(* IEC 61131-3 sources: AXOpen/src/integrations/app/src/Examples/AXOpen.AxoTask, 2 files *)

(* ---- AxoTaskDocuExample.st ---- *)
USING AXOpen.Core;

NAMESPACE AxoTaskExamples
    {S7.extern=ReadWrite}
    CLASS AxoTaskDocuExample EXTENDS  AXOpen.Core.AxoContext
        VAR PUBLIC
            {#ix-set:AttributeName = "<#Task name#>"}
            _myTask : AxoTask;
            _myCounter : ULINT;
        END_VAR

        METHOD PUBLIC Initialize
            // Initialization of the context needs to be called first
            // It does not need to be called cyclically, just once
            THIS.InitializeRootObject(_myTask);
        END_METHOD

        METHOD PROTECTED OVERRIDE Main
            THIS.InitializeRootObject(_myTask);
            // Cyclicall call of the Execute
            IF _myTask.Execute() THEN
                _myCounter := _myCounter + ULINT#1;
                _myTask.DoneWhen(_myCounter = ULINT#100);
            END_IF;
            IF _myTask.IsDone() THEN
                _myCounter := ULINT#0;
            END_IF;
        END_METHOD

        METHOD Examples
        //<AxoTaskInvokeDone>
            IF _myTask.Invoke().IsDone() THEN
                ; //Do something
            END_IF;
        //</AxoTaskInvokeDone>

        //<AxoTaskInvokeDoneSeparatelly>
            _myTask.Invoke();

            IF _myTask.IsDone() THEN
                ; //Do something
            END_IF;
        //</AxoTaskInvokeDoneSeparatelly>

        //<AxoTaskRunning>
             IF _myTask.Invoke().IsBusy() THEN
                ; //Do something
            END_IF;
        //</AxoTaskRunning>

        //<AxoTaskError>
            IF _myTask.Invoke().HasError() THEN
                ; //Do something
            END_IF;
        //</AxoTaskError>

        //<AxoTaskInvoke>
            _myTask.Invoke();
        //</AxoTaskInvoke>
        END_METHOD
    END_CLASS

    //<AxoTaskEventLikeMethods>
    {S7.extern=ReadWrite}
    CLASS MyTaskExample EXTENDS AXOpen.Core.AxoTask
        VAR
            OnAbortCounter : ULINT;
            OnResumeCounter : ULINT;
            OnDoneCounter : ULINT;
            OnErrorCounter : ULINT;
            OnRestoreCounter : ULINT;
            OnStartCounter : ULINT;
            WhileErrorCounter : ULINT;
        END_VAR
        METHOD PROTECTED OVERRIDE OnAbort
            OnAbortCounter := OnAbortCounter + ULINT#1;
        END_METHOD

        METHOD PROTECTED OVERRIDE OnResume
            OnResumeCounter := OnResumeCounter + ULINT#1;
        END_METHOD

        METHOD PROTECTED OVERRIDE OnDone
            OnDoneCounter := OnDoneCounter + ULINT#1;
        END_METHOD

        METHOD PROTECTED OVERRIDE OnError
            OnErrorCounter := OnErrorCounter + ULINT#1;
        END_METHOD

        METHOD PROTECTED OVERRIDE OnRestore
            OnRestoreCounter := OnRestoreCounter + ULINT#1;
        END_METHOD

        METHOD PROTECTED OVERRIDE OnStart
            OnStartCounter := OnStartCounter + ULINT#1;
        END_METHOD

        METHOD PROTECTED OVERRIDE WhileError
            WhileErrorCounter := WhileErrorCounter + ULINT#1;
        END_METHOD
    END_CLASS
    //</AxoTaskEventLikeMethods>
END_NAMESPACE

(* ---- AxoTaskExample.st ---- *)
USING AXOpen.Core;

NAMESPACE AxoTaskExamples

    {S7.extern=ReadWrite}
    CLASS MyCommandTask EXTENDS AXOpen.Core.AxoTask
        VAR PUBLIC
        {#ix-set:AttributeName = "<#Counter#>"}
        _counter : ULINT;
        END_VAR

        METHOD PROTECTED OVERRIDE OnRestore
            _counter := ULINT#0;
        END_METHOD
    END_CLASS

    {S7.extern=ReadWrite}
    CLASS Tasks EXTENDS AXOpen.Core.AxoContext
        VAR PUBLIC
            {#ix-set:AttributeName = "Click to execute this command"}
            _commandTask : MyCommandTask;
            {#ix-set:AttributeName = "If true the command will end in failure."}
            _commandEndsInFailure : BOOL;
        END_VAR

        METHOD PROTECTED OVERRIDE Main
            THIS.InitializeRootObject(_commandTask);

            IF(_commandTask.Execute()) THEN
                _commandTask._counter := _commandTask._counter + ULINT#1;
                IF (_commandTask._counter MOD ULINT#250) = ULINT#0 THEN
                    IF(_commandEndsInFailure) THEN
                        _commandTask.ThrowWhen(TRUE);
                    ELSE
                        _commandTask.DoneWhen(TRUE);
                    END_IF;
                END_IF;
            END_IF;
        END_METHOD
    END_CLASS
END_NAMESPACE
